FUNCTION_BLOCK TestECC
  (* Version 1.0, 2008-04-21, Goran Cengic, Chalmers *)
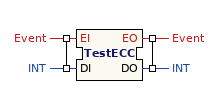
  EVENT_INPUT
    EI WITH DI;
  END_EVENT
  EVENT_OUTPUT
    EO WITH DO;
  END_EVENT
  VAR_INPUT
    DI : INT;
  END_VAR
  VAR_OUTPUT
    DO : INT;
  END_VAR
  VAR
    invoked : INT;
  END_VAR
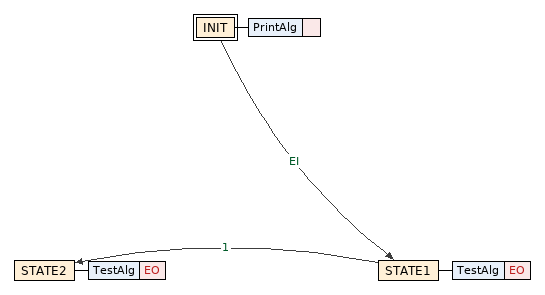
  EC_STATES
    INIT : PrintAlg;
    STATE1 : TestAlg -> EO;
    STATE2 : TestAlg -> EO;
  END_STATES
  EC_TRANSITIONS
    INIT TO STATE1 := EI;
    STATE1 TO STATE2 := 1;
  END_TRANSITIONS
  ALGORITHM TestAlg IN Java:
invoked = invoked + 1;
	DO = DI + 1;
	System.out.println("TestAlg:invoked: " + invoked + " times.");
	System.out.println("TestAlg: DO: " + DO + ".");
  END_ALGORITHM
  ALGORITHM PrintAlg IN Java:
System.out.println("InitAlg:invoked: " + invoked + " times.");
	System.out.println("InitAlg: DO: " + DO + ".");
  END_ALGORITHM
END_FUNCTION_BLOCK
